FUNCTION_BLOCK MAX_INT (* IEC 61131-3 INT Maximum *)
  (* Standard: 61131-3 *)
  (* Version 0.0, 2004-12-15, JHC, Rockwell Automation, Converted from SRC format. *)
  (* Compiler header: package fb.rt.plc.select; *)
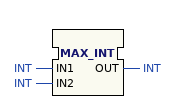
  VAR_INPUT
    IN1 : INT;
    IN2 : INT;
  END_VAR
  VAR_OUTPUT
    OUT : INT; (* MAX(IN1,IN2) *)
  END_VAR
END_FUNCTION_BLOCK
